(*

short summary
=============
dispather for cramel candy

legal notes
===========
SPDX-FileCopyrightText: © 2024 ekvip automation GmbH <info@ekvip.de>
SPDX-License-Identifier: Apache-2.0
For details check: Apache-2.0_

.. _Apache-2.0: https://www.apache.org/licenses/LICENSE-2.0

*)

{attribute 'enable_dynamic_creation'}
FUNCTION_BLOCK FINAL CaramelCandyDispatcher EXTENDS AbstractCandyDispatcher

(*

short summary
=============
this method dispatches caramel candies
to a candy consumer 

legal notes
===========
SPDX-FileCopyrightText: © 2024 ekvip automation GmbH <info@ekvip.de>
SPDX-License-Identifier: Apache-2.0
For details check: Apache-2.0_

.. _Apache-2.0: https://www.apache.org/licenses/LICENSE-2.0

*)

METHOD eat
VAR_INPUT
	(* consumer who eats the candy *)
	consumer	:REFERENCE TO AbstractCandyConsumer;
	(* candy amount in gram *)
	amount		:CandyAmountInGram;
END_VAR
RETURN(THIS^.eatCandiesIsImpossible(consumer, amount));
consumer.eatCaramelCandy(amount);
END_METHOD

END_FUNCTION_BLOCK

(* stored: Version 1.1.0.1
   POU CaramelCandyDispatcher: Id {114e7563-6e20-41bf-8a86-763f199435d8}, SpecialFunc None
   Method eat: Id {5d9d60c1-d2e6-4a51-868a-18cdd2858d16} *)
